# B&R Automation Studio project FrameworkTestStart
Automation Studio 4.10.3.60 SP; technology packages: mappView 5.16.1

## Configuration Config1

CPU X20CP1586, AutomationRuntime B4.91, Build 4.1.2, Safety 0.0, Vc V4.62.0

### Task classes (Cpu.sw)
```
Cyclic#4:
  Program <- Program.prg
Libraries: McBase, CoTrace, AsZip, FileIO, runtime
```

### Hardware
```
X20CP1586 : X20CP1586 v1.9.0.0
  Connector IF1:
    ActivateIna = 0
  Connector IF2:
    ActivateDevice = 1
    Mode = Manual
    InternetAddress = 192.168.0.20
    SubnetMask = 255.255.255.0
    InaPort = 11160
    ActivateSnmp = 2
  ConfigurationID = MVtest_Config1
  UserPartitionSize = 0
  Simulation = 1
  FileDevice1
  FileDeviceName1 = USER
  FileDevicePath1 = USER_PATH
  ActivateOpcUa = 1
  OpcUaInformationModels_PV_Version = 1
```

- Safety project (password-protected, skipped)

## Logical view

Binary libraries used (declarations not repeated): operator, runtime, astime, AsIecCon, AsZip, FileIO, McBase, CoTrace 5.16.0

### Package Logical/Libraries - Global libraries

- Visualisation Logical/mappView (not shown)

### Program Logical/Program (IEC)

#### Main.st - Init, cyclic, exit code
```iecst
PROGRAM _INIT
	testINT;
	testSTRING;
	testBOOL;

END_PROGRAM

PROGRAM _CYCLIC
	(* Insert code here *)

END_PROGRAM

PROGRAM _EXIT
	(* Insert code here *)

END_PROGRAM
```

#### Variables.var - Local variables
```iecst
VAR
	testINT : INT;
	testSTRING : STRING[80];
	testBOOL : BOOL;
END_VAR
```

Listed in the project but not available here: Logical/Global.typ, Logical/Global.var, Logical/Program/Types.typ
